// TIA Portal V20 export
TYPE "LER_typeCount"
// stored: Access Published
   STRUCT
      CountPV : Int;
      CountSV : Int;
   END_STRUCT;
END_TYPE
